{region '#Template'}
	{attribute 'Version' := '5.1.0.0'}
	{attribute 'Tags' := '"LCID": "1031", "Text": "Gewerk, Gebäudeautomation, Daten"'}
	{attribute 'Tags' := '"LCID": "1033", "Text": "Trade, Building automation, data"'}
	{attribute 'Using' := '"Type": "Template", "URI": "Site"'}
	{attribute 'Description' := '"LCID": "1031", "Text": "Aufruf der Aggregate der allgemeinen Gebäudedaten"'}
	{attribute 'Description' := '"LCID": "1033", "Text": "Calling the aggrgates of common building data"'}
{endregion}	 
FUNCTION_BLOCK FB_BA_BuildingData EXTENDS FB_BA_View
VAR_INPUT
END_VAR
VAR_OUTPUT
END_VAR
VAR_INPUT CONSTANT
	BuildingEnergLvl			: FB_BA_BuildingEnergyLevel;
	BuildingSpRmT				: FB_BA_BuildingSpRmT;
END_VAR
VAR
END_VAR

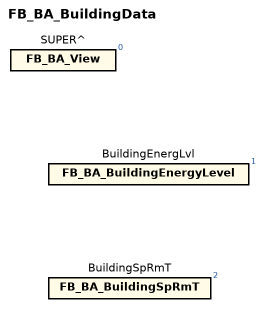
SUPER^(); // FB_BA_View
BuildingEnergLvl(); // FB_BA_BuildingEnergyLevel
BuildingSpRmT(); // FB_BA_BuildingSpRmT

METHOD FB_init : BOOL
VAR_INPUT
	bInitRetains : BOOL; // if TRUE, the retain variables are initialized (warm start / cold start)
	bInCopyCode : BOOL;  // if TRUE, the instance afterwards gets moved into the copy code (online change)
END_VAR
BuildingEnergLvl.iParent		:= THIS^;	
BuildingEnergLvl.iLabel			:= LblCtl_BuildingEnergyLevel;  
BuildingEnergLvl.sObjectName	:= '{Idx=01}';
BuildingEnergLvl.eDPADMode		:= E_BA_DPADMode.eInclude;

BuildingSpRmT.iParent			:= THIS^;	
BuildingSpRmT.iLabel			:= LblCtl_BuildingSpRmT;  
BuildingSpRmT.sObjectName		:= '{Idx=02}';
BuildingSpRmT.eDPADMode			:= E_BA_DPADMode.eInclude;
END_METHOD

END_FUNCTION_BLOCK

(* stored: Version 1.1.0.1, ProductVersion 3.1.4024.12
   POU FB_BA_BuildingData: Id {6b4af8a1-c69a-4446-861d-dedff3625df1}, SpecialFunc None
   Method FB_init: Id {345b4860-156d-483c-80c7-f3741dafe595} *)
